FUNCTION_BLOCK ConveyorSC_NC
VAR_INPUT
	bEnable : BOOL;
END_VAR
VAR_OUTPUT
	sensorEntry AT %I* : BOOL := TRUE;
	sensorExit AT %I* : BOOL := TRUE;
	
	trueMode : ConveyorMode;
	requestedMode : ConveyorMode;
	
	position : LREAL;
	velocity : LREAL;
	ready : BOOL;
END_VAR
VAR
	axis : AXIS_REF;
	
	mcReadPosition : MC_ReadActualPosition; //continuous enable FBs
	mcReadVelocity : MC_ReadActualVelocity;
	mcReadError : MC_ReadAxisError;
	mcPower : MC_Power;
	
	mcReset : MC_Reset; //rising edge FBs
	mcMoveAbsolute : MC_MoveAbsolute;
	mcMoveRelative : MC_MoveRelative;
	mcMoveVelocity : MC_MoveVelocity;
	
	mcSetPosition : MC_SetPosition;
	mcStop : MC_Stop;
END_VAR
VAR_STAT CONSTANT
	targetingVelocity : INT := 500;
	continuousVelocity : INT := 500;
END_VAR
(*
this FB represents a standard slat conveyor with no lifter
	compliant with PLCopen motion control

unlike standalone servos,
	conveyors need to coordinate (not slave) their motion with other conveyors
	and be able to set their current position to any value as required by the system
	
moveAbsolute is provided for now but should not be used for position targetting and may be protected/privated later
instead, request/set the operation mode and the motion will follow
*)

IF error THEN
	stop();
	reset();
	
ELSE
	CASE trueMode OF
		ConveyorMode.IDLE:			stop();	
		ConveyorMode.FORWARD:		moveContinuous(direction:= MC_Positive_Direction);
		ConveyorMode.BACKWARD:		moveContinuous(direction:= MC_Negative_Direction);
		ConveyorMode.STOP:			stop();
	END_CASE
	
END_IF

blocks();

mcReset.Execute := FALSE;
mcMoveAbsolute.Execute := FALSE;
mcMoveRelative.Execute := FALSE;
mcMoveVelocity.Execute := FALSE;
mcSetPosition.Execute := FALSE;
mcStop.Execute := FALSE;

blocks();

PROPERTY Active : BOOL
GET
Active := 
	mcMoveAbsolute.Busy OR 
	mcMoveRelative.Busy OR 
	mcMoveVelocity.Busy OR 
	mcSetPosition.Busy OR 
	mcReset.Busy OR 
	mcStop.Busy;
END_GET
END_PROPERTY

METHOD PRIVATE blocks : BOOL
mcReadPosition(
	Axis:= axis, 
	Enable:= TRUE, 
	Valid=> , 
	Busy=> , 
	Error=> , 
	ErrorID=> , 
	Position=> position);
	
mcReadVelocity(
	Axis:= axis, 
	Enable:= TRUE, 
	Valid=> , 
	Busy=> , 
	Error=> , 
	ErrorID=> , 
	ActualVelocity=> velocity);
	
mcReadError(
	Axis:= axis, 
	Enable:= TRUE, 
	Valid=> , 
	Busy=> , 
	Error=> , 
	ErrorID=> , 
	AxisErrorID=> );
	
mcPower(
	Axis:= axis, 
	Enable:= bEnable, 
	Enable_Positive:= TRUE, 
	Enable_Negative:= TRUE, 
	Override:= 100, 
	BufferMode:= , 
	Options:= , 
	Status=> , 
	Busy=> , 
	Active=> , 
	Error=> , 
	ErrorID=> );

mcReset(
	Axis:= axis, 
	Execute:= , 
	Done=> , 
	Busy=> , 
	Error=> , 
	ErrorID=> );

mcMoveAbsolute(
	Axis:= axis, 
	Execute:= , 
	Position:= , 
	Velocity:= targetingVelocity, 
	Acceleration:= , 
	Deceleration:= , 
	Jerk:= , 
	BufferMode:= , 
	Options:= , 
	Done=> , 
	Busy=> , 
	Active=> , 
	CommandAborted=> , 
	Error=> , 
	ErrorID=> );
	
mcMoveRelative(
	Axis:= axis, 
	Execute:= , 
	Distance:= ,
	Velocity:= targetingVelocity, 
	Acceleration:= , 
	Deceleration:= , 
	Jerk:= , 
	BufferMode:= , 
	Options:= , 
	Done=> , 
	Busy=> , 
	Active=> , 
	CommandAborted=> , 
	Error=> , 
	ErrorID=> );
	
mcMoveVelocity( //stopped with stop();
	Axis:= axis, 
	Execute:= , 
	Velocity:= continuousVelocity, 
	Acceleration:= , 
	Deceleration:= , 
	Jerk:= , 
	Direction:= , 
	BufferMode:= , 
	Options:= , 
	InVelocity=> , 
	Busy=> , 
	Active=> , 
	CommandAborted=> , 
	Error=> , 
	ErrorID=> );
	
mcSetPosition(
	Axis:= axis, 
	Execute:= , 
	Position:= , 
	Mode:= , 
	Options:= , 
	Done=> , 
	Busy=> , 
	Error=> , 
	ErrorID=> );
	
mcStop(
	Axis:= axis, 
	Execute:= , 
	Deceleration:= , 
	Jerk:= , 
	Options:= , 
	Done=> , 
	Busy=> , 
	Active=> , 
	CommandAborted=> , 
	Error=> , 
	ErrorID=> );
END_METHOD

PROPERTY CurrentPosition : LREAL
GET
CurrentPosition := position;
END_GET
SET
position := CurrentPosition;
END_SET
END_PROPERTY

PROPERTY Error : BOOL
GET
error := 
	mcMoveAbsolute.Error OR 
	mcMoveRelative.Error OR 
	mcMoveVelocity.Error OR 
	mcSetPosition.Error OR 
	mcReset.Error OR 
	mcStop.Error OR
	mcReadError.AxisErrorID > 0;
END_GET
END_PROPERTY

{attribute 'monitoring' := 'call'}
PROPERTY IsOccupied : BOOL
GET
IsOccupied := sensorExit OR sensorEntry;
END_GET
END_PROPERTY

METHOD moveAbsolute : BOOL
VAR_INPUT
	newTarget : REAL;
END_VAR
mcMoveAbsolute.Position := newTarget;

IF NOT Active AND NOT error THEN
	mcMoveAbsolute.Execute := TRUE;
END_IF

moveAbsolute := 
	//mcMoveAbsolute.Done;
	CurrentPosition = TargetPosition;
END_METHOD

METHOD moveContinuous : BOOL
VAR_INPUT
	direction : MC_Direction;
END_VAR
mcMoveVelocity.Direction := direction;

IF NOT Active AND NOT error THEN
	mcMoveVelocity.Execute := TRUE;
	moveContinuous := TRUE;
END_IF
END_METHOD

METHOD reset : BOOL
VAR_INPUT
END_VAR
mcReset.Execute := TRUE;

reset := mcReset.Done;
END_METHOD

METHOD setMode : BOOL
VAR_INPUT
	mode : ConveyorMode;
END_VAR
trueMode := mode;
END_METHOD

METHOD setRequest : BOOL
VAR_INPUT
	newRequest : ConveyorMode;
END_VAR
requestedMode := newRequest;
END_METHOD

METHOD stop : BOOL
VAR_INPUT
END_VAR
mcStop.Execute := TRUE;

mcMoveAbsolute.Execute := FALSE;
mcMoveRelative.Execute := FALSE;
mcMoveVelocity.Execute := FALSE;
END_METHOD

PROPERTY TargetPosition : LREAL
GET
END_GET
SET
moveAbsolute(newTarget := TargetPosition);
END_SET
END_PROPERTY

END_FUNCTION_BLOCK

(* stored: Version 1.1.0.1, ProductVersion 3.1.4024.11
   POU ConveyorSC_NC: Id {42eb6a02-0556-427e-a01f-090cd2356560}, SpecialFunc None
   Folder OpMode: Id {d08f0925-1051-460e-b699-f68626ae491a}
   Folder Private: Id {c1ceb5d7-45c2-4dba-a5a5-f2345a352849}
   Folder Properties: Id {ac48330c-bd0c-4df0-aae5-eb8c4e9b2a04}
   Property Active: Id {b9846c9d-0973-4916-a809-828e8bac60a1}
   Get Get: Id {ab644ead-161c-4918-bb39-bf9d10d2deac}
   Method blocks: Id {1e6a7e8e-22f1-47c6-a60d-2dd68d62435a}
   Property CurrentPosition: Id {0cf081fd-2188-46f2-8270-9c17a4944e39}
   Get Get: Id {8f3dbf7b-0535-4418-b3ba-b30d720bf456}
   Set Set: Id {00fe20ed-4207-470d-965c-4c23fb230144}
   Property Error: Id {17949c08-c0bf-41ef-bbc6-5c7512a312ee}
   Get Get: Id {05305283-5e7a-42ce-9f39-02b3a802344d}
   Property IsOccupied: Id {ba8708dd-a466-428c-915c-8331ed048fb6}
   Get Get: Id {d2f452a1-a21b-43fd-8a24-47b5f82bd7fb}
   Method moveAbsolute: Id {c0a3facf-01a6-4fa9-838e-e995e92b9c94}
   Method moveContinuous: Id {478a39e7-1e41-4b59-bc73-67d5f0d90925}
   Method reset: Id {6111573b-0260-4437-99d7-85339ca8130a}
   Method setMode: Id {f272a596-1e67-4bba-8c36-60ce98f5285a}
   Method setRequest: Id {9688c985-e44f-4288-91e2-b4e839e49609}
   Method stop: Id {2153e19f-9e1a-430b-9392-9f8b157e93fb}
   Property TargetPosition: Id {3cbbc18b-4e14-46ed-9728-52834e89fa82}
   Get Get: Id {7b0ae11d-e011-483c-83ff-400bf13fdcc9}
   Set Set: Id {0afd26bb-a492-4448-b2b6-22b01e223ffe} *)
